                                        FB_Bacnet.StartStopCommand_016.bEnWrite := TRUE;
                                        FB_Bacnet.StartStopCommand_016.bVal := TRUE;
                                    18: 
                                        
                                        FB_Bacnet.StartStopCommand_017.bEnWrite := TRUE;
                                        FB_Bacnet.StartStopCommand_017.bVal := TRUE;
                                    19: 
                                        
                                        FB_Bacnet.StartStopCommand_019.bEnWrite := TRUE;
                                        FB_Bacnet.StartStopCommand_019.bVal := TRUE;
                                    20:
                                        
                                        FB_Bacnet.StartStopCommand_018.bEnWrite := TRUE;
                                        FB_Bacnet.StartStopCommand_018.bVal := TRUE;
                                END_CASE
                            END_IF
                        END_FOR        
                    END_IF
                    // Schedule Unit OFF
                    IF wSchedWEHourEndFG_ = currH AND wSchedWEMinEndFG_ = currM AND NOT bUnitTriggered THEN
                        bUnitTriggered := TRUE;
                        FOR i := 1 TO 20 DO
                            // Send command unit OFF
                            IF bUnitFG_[i] THEN 
                                CASE i OF
                                    1: 
                                        
                                        FB_Bacnet.StartStopCommand_000.bEnWrite := TRUE;
                                        FB_Bacnet.StartStopCommand_000.bVal := FALSE;
                                    2: 
                                        
                                        FB_Bacnet.StartStopCommand_001.bEnWrite := TRUE;
                                        FB_Bacnet.StartStopCommand_001.bVal := FALSE;
                                    3: 
                                        
                                        FB_Bacnet.StartStopCommand_002.bEnWrite := TRUE;
                                        FB_Bacnet.StartStopCommand_002.bVal := FALSE;
                                    4: 
                                        
                                        FB_Bacnet.StartStopCommand_003.bEnWrite := TRUE;
                                        FB_Bacnet.StartStopCommand_003.bVal := FALSE;
                                    5: 
                                        
                                        FB_Bacnet.StartStopCommand_004.bEnWrite := TRUE;
                                        FB_Bacnet.StartStopCommand_004.bVal := FALSE;
                                    6: 
                                        
                                        FB_Bacnet.StartStopCommand_005.bEnWrite := TRUE;
                                        FB_Bacnet.StartStopCommand_005.bVal := FALSE;
                                    7: 
                                        
                                        FB_Bacnet.StartStopCommand_006.bEnWrite := TRUE;
                                        FB_Bacnet.StartStopCommand_006.bVal := FALSE;
                                    8: 
                                        
                                        FB_Bacnet.StartStopCommand_007.bEnWrite := TRUE;
                                        FB_Bacnet.StartStopCommand_007.bVal := FALSE;
                                    9: 
                                        
                                        FB_Bacnet.StartStopCommand_008.bEnWrite := TRUE;
                                        FB_Bacnet.StartStopCommand_008.bVal := FALSE;
                                    10: 
                                        
                                        FB_Bacnet.StartStopCommand_009.bEnWrite := TRUE;
                                        FB_Bacnet.StartStopCommand_009.bVal := FALSE;
                                    11: 
                                        
                                        FB_Bacnet.StartStopCommand_010.bEnWrite := TRUE;
                                        FB_Bacnet.StartStopCommand_010.bVal := FALSE;
                                    12: 
                                        
                                        FB_Bacnet.StartStopCommand_011.bEnWrite := TRUE;
                                        FB_Bacnet.StartStopCommand_011.bVal := FALSE;
                                    13: 
                                        
                                        FB_Bacnet.StartStopCommand_012.bEnWrite := TRUE;
                                        FB_Bacnet.StartStopCommand_012.bVal := FALSE;
                                    14: 
                                        
                                        FB_Bacnet.StartStopCommand_013.bEnWrite := TRUE;
                                        FB_Bacnet.StartStopCommand_013.bVal := FALSE;
                                    15: 
                                        
                                        FB_Bacnet.StartStopCommand_014.bEnWrite := TRUE;
                                        FB_Bacnet.StartStopCommand_014.bVal := FALSE;
                                    16: 
                                        
                                        FB_Bacnet.StartStopCommand_015.bEnWrite := TRUE;
                                        FB_Bacnet.StartStopCommand_015.bVal := FALSE;
                                    17: 
                                        
                                        FB_Bacnet.StartStopCommand_016.bEnWrite := TRUE;
                                        FB_Bacnet.StartStopCommand_016.bVal := FALSE;
                                    18: 
                                        
                                        FB_Bacnet.StartStopCommand_017.bEnWrite := TRUE;
                                        FB_Bacnet.StartStopCommand_017.bVal := FALSE;
                                    19: 
                                        
                                        FB_Bacnet.StartStopCommand_019.bEnWrite := TRUE;
                                        FB_Bacnet.StartStopCommand_019.bVal := FALSE;
                                    20:
                                        
                                        FB_Bacnet.StartStopCommand_018.bEnWrite := TRUE;
                                        FB_Bacnet.StartStopCommand_018.bVal := FALSE;
                                END_CASE
                            END_IF
                        END_FOR
                    END_IF
                END_IF
            END_IF
        END_IF

END_FUNCTION_BLOCK

// ---- POUs/FB_Scheduler/FB_Scheduler_FB2.TcPOU

      FUNCTION_BLOCK FB_Scheduler_FB2
      VAR_INPUT
          currH : WORD;
          currM : WORD;
          currD : WORD;
      END_VAR
      VAR_IN_OUT
          FB_Bacnet : FB_BACnet_DAIKIN_MasterStation_III_No_1;
      END_VAR
      VAR
          i : INT;
          bUnitTriggered : BOOL := FALSE; // New flag to track execution
          prevMinute : WORD := 0;        // New variable to track the previous minute
      END_VAR
      VAR PERSISTENT
          //scheduler var
          bEnSchedFB2_ : BOOL;
          wSchedWDHourStartFB2_ : WORD; 
          wSchedWDMinStartFB2_ : WORD; 
          wSchedWEHourStartFB2_ : WORD; 
          wSchedWEMinStartFB2_ : WORD;
          wSchedWDHourEndFB2_ : WORD;
          wSchedWDMinEndFB2_ : WORD;
          wSchedWEHourEndFB2_ : WORD;
          wSchedWEMinEndFB2_ : WORD;
          //unit var
          bUnitFB2_ : ARRAY [1..13] OF BOOL;
      END_VAR


        // Reset trigger flag at minute change or at the exact scheduled time
        IF currM <> prevMinute OR 
           (currH = wSchedWDHourStartFB2_ AND currM = wSchedWDMinStartFB2_) OR 
           (currH = wSchedWDHourEndFB2_ AND currM = wSchedWDMinEndFB2_) THEN
            bUnitTriggered := FALSE;
            prevMinute := currM;
        END_IF

        // Unit Schedule Enable
        IF bEnSchedFB2_ THEN
            // Weekday schedule
            IF currD >= 1 AND currD <= 5 THEN
                IF (wSchedWDHourStartFB2_ <> wSchedWDHourEndFB2_ OR wSchedWDMinStartFB2_ <> wSchedWDMinEndFB2_) THEN
                    // Schedule Unit ON
                    IF wSchedWDHourStartFB2_ = currH AND wSchedWDMinStartFB2_ = currM AND NOT bUnitTriggered THEN
                        bUnitTriggered := TRUE;
                        FOR i := 1 TO 13 DO
                            // Send command unit ON
                            IF bUnitFB2_[i] THEN 
                                CASE i OF
                                    1: 
                                        
                                        FB_Bacnet.StartStopCommand_037.bEnWrite := TRUE;
                                        FB_Bacnet.StartStopCommand_037.bVal := TRUE;
                                    2: 
                                        
                                        FB_Bacnet.StartStopCommand_038.bEnWrite := TRUE;
                                        FB_Bacnet.StartStopCommand_038.bVal := TRUE;
                                    3: 
                                        
                                        FB_Bacnet.StartStopCommand_039.bEnWrite := TRUE;
                                        FB_Bacnet.StartStopCommand_039.bVal := TRUE;
                                    4: 
                                        //
                                        //FB_Bacnet.StartStopCommand_040.bEnWrite := TRUE;
                                        //FB_Bacnet.StartStopCommand_040.bVal := TRUE;
                                    5: 
                                        
                                        FB_Bacnet.StartStopCommand_041.bEnWrite := TRUE;
                                        FB_Bacnet.StartStopCommand_041.bVal := TRUE;
                                    6: 
                                        
                                        FB_Bacnet.StartStopCommand_042.bEnWrite := TRUE;
                                        FB_Bacnet.StartStopCommand_042.bVal := TRUE;
                                    7: 
                                        
                                        FB_Bacnet.StartStopCommand_043.bEnWrite := TRUE;
                                        FB_Bacnet.StartStopCommand_043.bVal := TRUE;
                                    8: 
                                        //
                                        //FB_Bacnet.StartStopCommand_044.bEnWrite := TRUE;
                                        //FB_Bacnet.StartStopCommand_044.bVal := TRUE;
                                    9: 
                                        
                                        FB_Bacnet.StartStopCommand_045.bEnWrite := TRUE;
                                        FB_Bacnet.StartStopCommand_045.bVal := TRUE;
                                    10: 
                                        
                                        FB_Bacnet.StartStopCommand_046.bEnWrite := TRUE;
                                        FB_Bacnet.StartStopCommand_046.bVal := TRUE;
                                    11: 
                                        //
                                        //FB_Bacnet.StartStopCommand_047.bEnWrite := TRUE;
                                        //FB_Bacnet.StartStopCommand_047.bVal := TRUE;
                                    12: 
                                        //
                                        //FB_Bacnet.StartStopCommand_048.bEnWrite := TRUE;
                                        //FB_Bacnet.StartStopCommand_048.bVal := TRUE;
                                    13: 
                                        
                                        FB_Bacnet.StartStopCommand_049.bEnWrite := TRUE;
                                        FB_Bacnet.StartStopCommand_049.bVal := TRUE;
                                END_CASE
                            END_IF
                        END_FOR
                    END_IF
                    // Schedule Unit OFF
                    IF wSchedWDHourEndFB2_ = currH AND wSchedWDMinEndFB2_ = currM AND NOT bUnitTriggered THEN
                        bUnitTriggered := TRUE;
                        FOR i := 1 TO 13 DO
                            // Send command unit OFF
                            IF bUnitFB2_[i] THEN 
                                CASE i OF
                                    1: 
                                        
                                        FB_Bacnet.StartStopCommand_037.bEnWrite := TRUE;
                                        FB_Bacnet.StartStopCommand_037.bVal := FALSE;
                                    2: 
                                        
                                        FB_Bacnet.StartStopCommand_038.bEnWrite := TRUE;
                                        FB_Bacnet.StartStopCommand_038.bVal := FALSE;
                                    3: 
                                        
                                        FB_Bacnet.StartStopCommand_039.bEnWrite := TRUE;
                                        FB_Bacnet.StartStopCommand_039.bVal := FALSE;
                                    4: 
                                        //
                                        //FB_Bacnet.StartStopCommand_040.bEnWrite := TRUE;
                                        //FB_Bacnet.StartStopCommand_040.bVal := FALSE;
                                    5: 
                                        
                                        FB_Bacnet.StartStopCommand_041.bEnWrite := TRUE;
                                        FB_Bacnet.StartStopCommand_041.bVal := FALSE;
                                    6: 
                                        
                                        FB_Bacnet.StartStopCommand_042.bEnWrite := TRUE;
                                        FB_Bacnet.StartStopCommand_042.bVal := FALSE;
                                    7: 
                                        
                                        FB_Bacnet.StartStopCommand_043.bEnWrite := TRUE;
                                        FB_Bacnet.StartStopCommand_043.bVal := FALSE;
                                    8: 
                                        //
                                        //FB_Bacnet.StartStopCommand_044.bEnWrite := TRUE;
                                        //FB_Bacnet.StartStopCommand_044.bVal := FALSE;
                                    9: 
                                        
                                        FB_Bacnet.StartStopCommand_045.bEnWrite := TRUE;
                                        FB_Bacnet.StartStopCommand_045.bVal := FALSE;
                                    10: 
                                        
                                        FB_Bacnet.StartStopCommand_046.bEnWrite := TRUE;
                                        FB_Bacnet.StartStopCommand_046.bVal := FALSE;
                                    11: 
                                        //
                                        //FB_Bacnet.StartStopCommand_047.bEnWrite := TRUE;
                                        //FB_Bacnet.StartStopCommand_047.bVal := FALSE;
                                    12: 
                                        //
                                        //FB_Bacnet.StartStopCommand_048.bEnWrite := TRUE;
                                        //FB_Bacnet.StartStopCommand_048.bVal := FALSE;
                                    13: 
                                        
                                        FB_Bacnet.StartStopCommand_049.bEnWrite := TRUE;
                                        FB_Bacnet.StartStopCommand_049.bVal := FALSE;
                                END_CASE
                            END_IF
                        END_FOR
                    END_IF
                END_IF
            END_IF

            // Weekend schedule
            IF currD = 0 OR currD = 6 THEN
                IF (wSchedWEHourStartFB2_ <> wSchedWEHourEndFB2_ OR wSchedWEMinStartFB2_ <> wSchedWEMinEndFB2_) THEN
                    // Schedule Unit ON
                    IF wSchedWEHourStartFB2_ = currH AND wSchedWEMinStartFB2_ = currM AND NOT bUnitTriggered THEN
                        bUnitTriggered := TRUE;
                        FOR i := 1 TO 13 DO
                            // Send command unit ON
                            IF bUnitFB2_[i] THEN 
                                CASE i OF
                                    1: 
                                        
                                        FB_Bacnet.StartStopCommand_037.bEnWrite := TRUE;
                                        FB_Bacnet.StartStopCommand_037.bVal := TRUE;
                                    2: 
                                        
                                        FB_Bacnet.StartStopCommand_038.bEnWrite := TRUE;
                                        FB_Bacnet.StartStopCommand_038.bVal := TRUE;
                                    3: 
                                        
                                        FB_Bacnet.StartStopCommand_039.bEnWrite := TRUE;
                                        FB_Bacnet.StartStopCommand_039.bVal := TRUE;
                                    4: 
                                        //
                                        //FB_Bacnet.StartStopCommand_040.bEnWrite := TRUE;
                                        //FB_Bacnet.StartStopCommand_040.bVal := TRUE;
                                    5: 
                                        
                                        FB_Bacnet.StartStopCommand_041.bEnWrite := TRUE;
                                        FB_Bacnet.StartStopCommand_041.bVal := TRUE;
                                    6: 
                                        
                                        FB_Bacnet.StartStopCommand_042.bEnWrite := TRUE;
                                        FB_Bacnet.StartStopCommand_042.bVal := TRUE;
                                    7: 
                                        
                                        FB_Bacnet.StartStopCommand_043.bEnWrite := TRUE;
                                        FB_Bacnet.StartStopCommand_043.bVal := TRUE;
                                    8: 
                                        //
                                        //FB_Bacnet.StartStopCommand_044.bEnWrite := TRUE;
                                        //FB_Bacnet.StartStopCommand_044.bVal := TRUE;
                                    9: 
                                        
                                        FB_Bacnet.StartStopCommand_045.bEnWrite := TRUE;
                                        FB_Bacnet.StartStopCommand_045.bVal := TRUE;
                                    10: 
                                        
                                        FB_Bacnet.StartStopCommand_046.bEnWrite := TRUE;
                                        FB_Bacnet.StartStopCommand_046.bVal := TRUE;
                                    11: 
                                        //
                                        //FB_Bacnet.StartStopCommand_047.bEnWrite := TRUE;
                                        //FB_Bacnet.StartStopCommand_047.bVal := TRUE;
                                    12: 
                                        //
                                        //FB_Bacnet.StartStopCommand_048.bEnWrite := TRUE;
                                        //FB_Bacnet.StartStopCommand_048.bVal := TRUE;
                                    13: 
                                        
                                        FB_Bacnet.StartStopCommand_049.bEnWrite := TRUE;
                                        FB_Bacnet.StartStopCommand_049.bVal := TRUE;
                                END_CASE
                            END_IF
                        END_FOR
                    END_IF
                    // Schedule Unit OFF
                    IF wSchedWEHourEndFB2_ = currH AND wSchedWEMinEndFB2_ = currM AND NOT bUnitTriggered THEN
                        bUnitTriggered := TRUE;
                        FOR i := 1 TO 13 DO
                            // Send command unit OFF
                            IF bUnitFB2_[i] THEN 
                                CASE i OF
                                    1: 
                                        
                                        FB_Bacnet.StartStopCommand_037.bEnWrite := TRUE;
                                        FB_Bacnet.StartStopCommand_037.bVal := FALSE;
                                    2: 
                                        
                                        FB_Bacnet.StartStopCommand_038.bEnWrite := TRUE;
                                        FB_Bacnet.StartStopCommand_038.bVal := FALSE;
                                    3: 
                                        
                                        FB_Bacnet.StartStopCommand_039.bEnWrite := TRUE;
                                        FB_Bacnet.StartStopCommand_039.bVal := FALSE;
                                    4: 
                                        //
                                        //FB_Bacnet.StartStopCommand_040.bEnWrite := TRUE;
                                        //FB_Bacnet.StartStopCommand_040.bVal := FALSE;
                                    5: 
                                        
                                        FB_Bacnet.StartStopCommand_041.bEnWrite := TRUE;
                                        FB_Bacnet.StartStopCommand_041.bVal := FALSE;
                                    6: 
                                        
                                        FB_Bacnet.StartStopCommand_042.bEnWrite := TRUE;
                                        FB_Bacnet.StartStopCommand_042.bVal := FALSE;
                                    7: 
                                        
                                        FB_Bacnet.StartStopCommand_043.bEnWrite := TRUE;
                                        FB_Bacnet.StartStopCommand_043.bVal := FALSE;
                                    8: 
                                        //
                                        //FB_Bacnet.StartStopCommand_044.bEnWrite := TRUE;
                                        //FB_Bacnet.StartStopCommand_044.bVal := FALSE;
                                    9: 
                                        
                                        FB_Bacnet.StartStopCommand_045.bEnWrite := TRUE;
                                        FB_Bacnet.StartStopCommand_045.bVal := FALSE;
                                    10: 
                                        
                                        FB_Bacnet.StartStopCommand_046.bEnWrite := TRUE;
                                        FB_Bacnet.StartStopCommand_046.bVal := FALSE;
                                    11: 
                                        //
                                        //FB_Bacnet.StartStopCommand_047.bEnWrite := TRUE;
                                        //FB_Bacnet.StartStopCommand_047.bVal := FALSE;
                                    12: 
                                        //
                                        //FB_Bacnet.StartStopCommand_048.bEnWrite := TRUE;
                                        //FB_Bacnet.StartStopCommand_048.bVal := FALSE;
                                    13: 
                                        
                                        FB_Bacnet.StartStopCommand_049.bEnWrite := TRUE;
                                        FB_Bacnet.StartStopCommand_049.bVal := FALSE;
                                END_CASE
                            END_IF
                        END_FOR
                    END_IF
                END_IF
            END_IF
        END_IF

END_FUNCTION_BLOCK

// ---- POUs/FB_Scheduler/FB_Scheduler_FB1.TcPOU

      FUNCTION_BLOCK FB_Scheduler_FB1
      VAR_INPUT
          currH : WORD;
          currM : WORD;
          currD : WORD;
      END_VAR
      VAR_IN_OUT
          FB_Bacnet : FB_BACnet_DAIKIN_MasterStation_III_No_1;
      END_VAR
      VAR
          i : INT;
          bUnitTriggered : BOOL := FALSE; // New flag to track execution
          prevMinute : WORD := 0;        // New variable to track the previous minute
      END_VAR
      VAR PERSISTENT
          //scheduler var
          bEnSchedFB1_ : BOOL := FALSE;
          wSchedWDHourStartFB1_ : WORD; 
          wSchedWDMinStartFB1_ : WORD; 
          wSchedWEHourStartFB1_ : WORD; 
          wSchedWEMinStartFB1_ : WORD;
          wSchedWDHourEndFB1_ : WORD;
          wSchedWDMinEndFB1_ : WORD;
          wSchedWEHourEndFB1_ : WORD;
          wSchedWEMinEndFB1_ : WORD;
          //unit var
          bUnitFB1_ : ARRAY [1..17] OF BOOL;
      END_VAR


        // Reset trigger flag at minute change or at the exact scheduled time
        IF currM <> prevMinute OR 
           (currH = wSchedWDHourStartFB1_ AND currM = wSchedWDMinStartFB1_) OR 
           (currH = wSchedWDHourEndFB1_ AND currM = wSchedWDMinEndFB1_) THEN
            bUnitTriggered := FALSE;
            prevMinute := currM;
        END_IF

        // Unit Schedule Enable
        IF bEnSchedFB1_ THEN
            // Weekday schedule
            IF currD >= 1 AND currD <= 5 THEN
                IF (wSchedWDHourStartFB1_ <> wSchedWDHourEndFB1_ OR wSchedWDMinStartFB1_ <> wSchedWDMinEndFB1_) THEN
                    // Schedule Unit ON
                    IF wSchedWDHourStartFB1_ = currH AND wSchedWDMinStartFB1_ = currM AND NOT bUnitTriggered THEN
                        bUnitTriggered := TRUE;
                        FOR i := 1 TO 17 DO
                            // Send command unit ON
                            IF bUnitFB1_[i] THEN 
                                CASE i OF
                                    1: 
                                        
                                        FB_Bacnet.StartStopCommand_020.bEnWrite := TRUE;
                                        FB_Bacnet.StartStopCommand_020.bVal := TRUE;
                                    2: 
                                        
                                        FB_Bacnet.StartStopCommand_021.bEnWrite := TRUE;
                                        FB_Bacnet.StartStopCommand_021.bVal := TRUE;
                                    3: 
                                        
                                        FB_Bacnet.StartStopCommand_022.bEnWrite := TRUE;
                                        FB_Bacnet.StartStopCommand_022.bVal := TRUE;
                                    4: 
                                        
                                        FB_Bacnet.StartStopCommand_023.bEnWrite := TRUE;
                                        FB_Bacnet.StartStopCommand_023.bVal := TRUE;
                                    5: 
                                        
                                        FB_Bacnet.StartStopCommand_024.bEnWrite := TRUE;
                                        FB_Bacnet.StartStopCommand_024.bVal := TRUE;
                                    6: 
                                        
                                        FB_Bacnet.StartStopCommand_025.bEnWrite := TRUE;
                                        FB_Bacnet.StartStopCommand_025.bVal := TRUE;
                                    7: 
                                        
                                        FB_Bacnet.StartStopCommand_026.bEnWrite := TRUE;
                                        FB_Bacnet.StartStopCommand_026.bVal := TRUE;
                                    8: 
                                        
                                        FB_Bacnet.StartStopCommand_027.bEnWrite := TRUE;
                                        FB_Bacnet.StartStopCommand_027.bVal := TRUE;
                                    9: 
                                        
                                        FB_Bacnet.StartStopCommand_028.bEnWrite := TRUE;
                                        FB_Bacnet.StartStopCommand_028.bVal := TRUE;
                                    10: 
                                        
                                        FB_Bacnet.StartStopCommand_029.bEnWrite := TRUE;
                                        FB_Bacnet.StartStopCommand_029.bVal := TRUE;
                                    11: 
                                        
                                        FB_Bacnet.StartStopCommand_030.bEnWrite := TRUE;
                                        FB_Bacnet.StartStopCommand_030.bVal := TRUE;
                                    12: 
                                        
                                        FB_Bacnet.StartStopCommand_031.bEnWrite := TRUE;
                                        FB_Bacnet.StartStopCommand_031.bVal := TRUE;
                                    13: 
                                        
                                        FB_Bacnet.StartStopCommand_032.bEnWrite := TRUE;
                                        FB_Bacnet.StartStopCommand_032.bVal := TRUE;
                                    14: 
                                        
                                        FB_Bacnet.StartStopCommand_033.bEnWrite := TRUE;
                                        FB_Bacnet.StartStopCommand_033.bVal := TRUE;
                                    15: 
                                        
                                        FB_Bacnet.StartStopCommand_034.bEnWrite := TRUE;
                                        FB_Bacnet.StartStopCommand_034.bVal := TRUE;
                                    16: 
                                        
                                        FB_Bacnet.StartStopCommand_035.bEnWrite := TRUE;
                                        FB_Bacnet.StartStopCommand_035.bVal := TRUE;
                                    17: 
                                        
                                        FB_Bacnet.StartStopCommand_036.bEnWrite := TRUE;
                                        FB_Bacnet.StartStopCommand_036.bVal := TRUE;
                                END_CASE
                            END_IF
                        END_FOR
                    END_IF
                    // Schedule Unit OFF
                    IF wSchedWDHourEndFB1_ = currH AND wSchedWDMinEndFB1_ = currM AND NOT bUnitTriggered THEN
                        bUnitTriggered := TRUE;
                        FOR i := 1 TO 17 DO
                            // Send command unit OFF
                            IF bUnitFB1_[i] THEN 
                                CASE i OF
                                    1: 
                                        
                                        FB_Bacnet.StartStopCommand_020.bEnWrite := TRUE;
                                        FB_Bacnet.StartStopCommand_020.bVal := FALSE;
                                    2: 
                                        
                                        FB_Bacnet.StartStopCommand_021.bEnWrite := TRUE;
                                        FB_Bacnet.StartStopCommand_021.bVal := FALSE;
                                    3: 
                                        
                                        FB_Bacnet.StartStopCommand_022.bEnWrite := TRUE;
                                        FB_Bacnet.StartStopCommand_022.bVal := FALSE;
                                    4: 
                                        
                                        FB_Bacnet.StartStopCommand_023.bEnWrite := TRUE;
                                        FB_Bacnet.StartStopCommand_023.bVal := FALSE;
                                    5: 
                                        
                                        FB_Bacnet.StartStopCommand_024.bEnWrite := TRUE;
                                        FB_Bacnet.StartStopCommand_024.bVal := FALSE;
                                    6: 
                                        
                                        FB_Bacnet.StartStopCommand_025.bEnWrite := TRUE;
                                        FB_Bacnet.StartStopCommand_025.bVal := FALSE;
                                    7: 
                                        
                                        FB_Bacnet.StartStopCommand_026.bEnWrite := TRUE;
                                        FB_Bacnet.StartStopCommand_026.bVal := FALSE;
                                    8: 
                                        
                                        FB_Bacnet.StartStopCommand_027.bEnWrite := TRUE;
                                        FB_Bacnet.StartStopCommand_027.bVal := FALSE;
                                    9: 
                                        
                                        FB_Bacnet.StartStopCommand_028.bEnWrite := TRUE;
                                        FB_Bacnet.StartStopCommand_028.bVal := FALSE;
                                    10: 
                                        
                                        FB_Bacnet.StartStopCommand_029.bEnWrite := TRUE;
                                        FB_Bacnet.StartStopCommand_029.bVal := FALSE;
                                    11: 
                                        
                                        FB_Bacnet.StartStopCommand_030.bEnWrite := TRUE;
                                        FB_Bacnet.StartStopCommand_030.bVal := FALSE;
                                    12: 
                                        
                                        FB_Bacnet.StartStopCommand_031.bEnWrite := TRUE;
                                        FB_Bacnet.StartStopCommand_031.bVal := FALSE;
                                    13: 
                                        
                                        FB_Bacnet.StartStopCommand_032.bEnWrite := TRUE;
                                        FB_Bacnet.StartStopCommand_032.bVal := FALSE;
                                    14: 
                                        
                                        FB_Bacnet.StartStopCommand_033.bEnWrite := TRUE;
                                        FB_Bacnet.StartStopCommand_033.bVal := FALSE;
                                    15: 
                                        
                                        FB_Bacnet.StartStopCommand_034.bEnWrite := TRUE;
                                        FB_Bacnet.StartStopCommand_034.bVal := FALSE;
                                    16: 
                                        
                                        FB_Bacnet.StartStopCommand_035.bEnWrite := TRUE;
                                        FB_Bacnet.StartStopCommand_035.bVal := FALSE;
                                    17: 
                                        
                                        FB_Bacnet.StartStopCommand_036.bEnWrite := TRUE;
                                        FB_Bacnet.StartStopCommand_036.bVal := FALSE;
                                END_CASE
                            END_IF
                        END_FOR
                    END_IF
                END_IF
            END_IF

            // Weekend schedule
            IF currD = 0 OR currD = 6 THEN
                IF (wSchedWEHourStartFB1_ <> wSchedWEHourEndFB1_ OR wSchedWEMinStartFB1_ <> wSchedWEMinEndFB1_) THEN
                    // Schedule Unit ON
                    IF wSchedWEHourStartFB1_ = currH AND wSchedWEMinStartFB1_ = currM AND NOT bUnitTriggered THEN
                        bUnitTriggered := TRUE;
                        FOR i := 1 TO 17 DO
                            // Send command unit ON
                            IF bUnitFB1_[i] THEN 
                                CASE i OF
                                    1: 
                                        
                                        FB_Bacnet.StartStopCommand_020.bEnWrite := TRUE;
                                        FB_Bacnet.StartStopCommand_020.bVal := TRUE;
                                    2: 
                                        
                                        FB_Bacnet.StartStopCommand_021.bEnWrite := TRUE;
                                        FB_Bacnet.StartStopCommand_021.bVal := TRUE;
                                    3: 
                                        
                                        FB_Bacnet.StartStopCommand_022.bEnWrite := TRUE;
                                        FB_Bacnet.StartStopCommand_022.bVal := TRUE;
                                    4: 
                                        
                                        FB_Bacnet.StartStopCommand_023.bEnWrite := TRUE;
                                        FB_Bacnet.StartStopCommand_023.bVal := TRUE;
                                    5: 
                                        
                                        FB_Bacnet.StartStopCommand_024.bEnWrite := TRUE;
                                        FB_Bacnet.StartStopCommand_024.bVal := TRUE;
                                    6: 
                                        
                                        FB_Bacnet.StartStopCommand_025.bEnWrite := TRUE;
                                        FB_Bacnet.StartStopCommand_025.bVal := TRUE;
                                    7: 
                                        
                                        FB_Bacnet.StartStopCommand_026.bEnWrite := TRUE;
                                        FB_Bacnet.StartStopCommand_026.bVal := TRUE;
                                    8: 
                                        
                                        FB_Bacnet.StartStopCommand_027.bEnWrite := TRUE;
                                        FB_Bacnet.StartStopCommand_027.bVal := TRUE;
                                    9: 
                                        
                                        FB_Bacnet.StartStopCommand_028.bEnWrite := TRUE;
                                        FB_Bacnet.StartStopCommand_028.bVal := TRUE;
                                    10: 
                                        
                                        FB_Bacnet.StartStopCommand_029.bEnWrite := TRUE;
                                        FB_Bacnet.StartStopCommand_029.bVal := TRUE;
                                    11: 
                                        
                                        FB_Bacnet.StartStopCommand_030.bEnWrite := TRUE;
                                        FB_Bacnet.StartStopCommand_030.bVal := TRUE;
                                    12: 
                                        
                                        FB_Bacnet.StartStopCommand_031.bEnWrite := TRUE;
                                        FB_Bacnet.StartStopCommand_031.bVal := TRUE;
                                    13: 
                                        
                                        FB_Bacnet.StartStopCommand_032.bEnWrite := TRUE;
                                        FB_Bacnet.StartStopCommand_032.bVal := TRUE;
                                    14: 
                                        
                                        FB_Bacnet.StartStopCommand_033.bEnWrite := TRUE;
                                        FB_Bacnet.StartStopCommand_033.bVal := TRUE;
                                    15: 
                                        
                                        FB_Bacnet.StartStopCommand_034.bEnWrite := TRUE;
                                        FB_Bacnet.StartStopCommand_034.bVal := TRUE;
                                    16: 
                                        
                                        FB_Bacnet.StartStopCommand_035.bEnWrite := TRUE;
                                        FB_Bacnet.StartStopCommand_035.bVal := TRUE;
                                    17: 
                                        
                                        FB_Bacnet.StartStopCommand_036.bEnWrite := TRUE;
                                        FB_Bacnet.StartStopCommand_036.bVal := TRUE;
                                END_CASE
                            END_IF
                        END_FOR
                    END_IF
                    // Schedule Unit OFF
                    IF wSchedWEHourEndFB1_ = currH AND wSchedWEMinEndFB1_ = currM AND NOT bUnitTriggered THEN
                        bUnitTriggered := TRUE;
                        FOR i := 1 TO 17 DO
                            // Send command unit OFF
                            IF bUnitFB1_[i] THEN 
                                CASE i OF
                                    1: 
                                        
                                        FB_Bacnet.StartStopCommand_020.bEnWrite := TRUE;
                                        FB_Bacnet.StartStopCommand_020.bVal := FALSE;
                                    2: 
                                        
                                        FB_Bacnet.StartStopCommand_021.bEnWrite := TRUE;
                                        FB_Bacnet.StartStopCommand_021.bVal := FALSE;
                                    3: 
                                        
                                        FB_Bacnet.StartStopCommand_022.bEnWrite := TRUE;
                                        FB_Bacnet.StartStopCommand_022.bVal := FALSE;
                                    4: 
                                        
                                        FB_Bacnet.StartStopCommand_023.bEnWrite := TRUE;
                                        FB_Bacnet.StartStopCommand_023.bVal := FALSE;
                                    5: 
                                        
                                        FB_Bacnet.StartStopCommand_024.bEnWrite := TRUE;
                                        FB_Bacnet.StartStopCommand_024.bVal := FALSE;
                                    6: 
                                        
                                        FB_Bacnet.StartStopCommand_025.bEnWrite := TRUE;
                                        FB_Bacnet.StartStopCommand_025.bVal := FALSE;
                                    7: 
                                        
                                        FB_Bacnet.StartStopCommand_026.bEnWrite := TRUE;
                                        FB_Bacnet.StartStopCommand_026.bVal := FALSE;
                                    8: 
                                        
                                        FB_Bacnet.StartStopCommand_027.bEnWrite := TRUE;
                                        FB_Bacnet.StartStopCommand_027.bVal := FALSE;
                                    9: 
                                        
                                        FB_Bacnet.StartStopCommand_028.bEnWrite := TRUE;
                                        FB_Bacnet.StartStopCommand_028.bVal := FALSE;
                                    10: 
                                        
                                        FB_Bacnet.StartStopCommand_029.bEnWrite := TRUE;
                                        FB_Bacnet.StartStopCommand_029.bVal := FALSE;
                                    11: 
                                        
                                        FB_Bacnet.StartStopCommand_030.bEnWrite := TRUE;
                                        FB_Bacnet.StartStopCommand_030.bVal := FALSE;
                                    12: 
                                        
                                        FB_Bacnet.StartStopCommand_031.bEnWrite := TRUE;
                                        FB_Bacnet.StartStopCommand_031.bVal := FALSE;
                                    13: 
                                        
                                        FB_Bacnet.StartStopCommand_032.bEnWrite := TRUE;
                                        FB_Bacnet.StartStopCommand_032.bVal := FALSE;
                                    14: 
                                        
                                        FB_Bacnet.StartStopCommand_033.bEnWrite := TRUE;
                                        FB_Bacnet.StartStopCommand_033.bVal := FALSE;
                                    15: 
                                        
                                        FB_Bacnet.StartStopCommand_034.bEnWrite := TRUE;
                                        FB_Bacnet.StartStopCommand_034.bVal := FALSE;
                                    16: 
                                        
                                        FB_Bacnet.StartStopCommand_035.bEnWrite := TRUE;
                                        FB_Bacnet.StartStopCommand_035.bVal := FALSE;
                                    17: 
                                        
                                        FB_Bacnet.StartStopCommand_036.bEnWrite := TRUE;
                                        FB_Bacnet.StartStopCommand_036.bVal := FALSE;
                                END_CASE
                            END_IF
                        END_FOR
                    END_IF
                END_IF
            END_IF
        END_IF

END_FUNCTION_BLOCK

// ---- POUs/FB_Scheduler/FB_Scheduler_FMZ.TcPOU

      FUNCTION_BLOCK FB_Scheduler_FMZ
      VAR_INPUT
          currH : WORD;
          currM : WORD;
          currD : WORD;
      END_VAR
      VAR_IN_OUT
          FB_Bacnet : FB_BACnet_DAIKIN_MasterStation_III_No_1;
      END_VAR
      VAR
          i : INT;
          bUnitTriggered : BOOL := FALSE; // Flag to track execution
          prevMinute : WORD := 0;        // Track previous minute
      END_VAR
      VAR PERSISTENT
          //scheduler var
          bEnSchedFMZ_ : BOOL := FALSE;
          wSchedWDHourStartFMZ_ : WORD; 
          wSchedWDMinStartFMZ_ : WORD; 
          wSchedWEHourStartFMZ_ : WORD; 
          wSchedWEMinStartFMZ_ : WORD;
          wSchedWDHourEndFMZ_ : WORD;
          wSchedWDMinEndFMZ_ : WORD; 
          wSchedWEHourEndFMZ_ : WORD; 
          wSchedWEMinEndFMZ_ : WORD;
          //unit var
          bUnitFMZ_ : ARRAY [1..21] OF BOOL;
      END_VAR


        // Reset trigger flag at minute change or at the exact scheduled time
        IF currM <> prevMinute OR 
           (currH = wSchedWDHourStartFMZ_ AND currM = wSchedWDMinStartFMZ_) OR 
           (currH = wSchedWDHourEndFMZ_ AND currM = wSchedWDMinEndFMZ_) THEN
            bUnitTriggered := FALSE;
            prevMinute := currM;
        END_IF

        // Unit Schedule Enable
        IF bEnSchedFMZ_ THEN
            // Weekday schedule
            IF currD >= 1 AND currD <= 5 THEN
                IF (wSchedWDHourStartFMZ_ <> wSchedWDHourEndFMZ_ OR wSchedWDMinStartFMZ_ <> wSchedWDMinEndFMZ_) THEN
                    // Schedule Unit ON
                    IF wSchedWDHourStartFMZ_ = currH AND wSchedWDMinStartFMZ_ = currM AND NOT bUnitTriggered THEN
                        bUnitTriggered := TRUE;
                        FOR i := 1 TO 21 DO
                            // Send command unit ON
                            IF bUnitFMZ_[i] THEN 
                                CASE i OF
                                    1: 
                                        
                                        FB_Bacnet.StartStopCommand_064.bEnWrite := TRUE;
                                        FB_Bacnet.StartStopCommand_064.bVal := TRUE;
                                    2: 
                                        
                                        FB_Bacnet.StartStopCommand_065.bEnWrite := TRUE;
                                        FB_Bacnet.StartStopCommand_065.bVal := TRUE;
                                    3: 
                                        
                                        FB_Bacnet.StartStopCommand_066.bEnWrite := TRUE;
                                        FB_Bacnet.StartStopCommand_066.bVal := TRUE;
                                    4: 
                                        
                                        FB_Bacnet.StartStopCommand_067.bEnWrite := TRUE;
                                        FB_Bacnet.StartStopCommand_067.bVal := TRUE;
                                    5: 
                                        
                                        FB_Bacnet.StartStopCommand_068.bEnWrite := TRUE;
                                        FB_Bacnet.StartStopCommand_068.bVal := TRUE;
                                    6: 
                                        
                                        FB_Bacnet.StartStopCommand_069.bEnWrite := TRUE;
                                        FB_Bacnet.StartStopCommand_069.bVal := TRUE;
                                    7: 
                                        
                                        FB_Bacnet.StartStopCommand_070.bEnWrite := TRUE;
                                        FB_Bacnet.StartStopCommand_070.bVal := TRUE;
                                    8: 
                                        
                                        FB_Bacnet.StartStopCommand_071.bEnWrite := TRUE;
                                        FB_Bacnet.StartStopCommand_071.bVal := TRUE;
                                    9: 
                                        
                                        FB_Bacnet.StartStopCommand_072.bEnWrite := TRUE;
                                        FB_Bacnet.StartStopCommand_072.bVal := TRUE;
                                    10: 
                                        
                                        FB_Bacnet.StartStopCommand_073.bEnWrite := TRUE;
                                        FB_Bacnet.StartStopCommand_073.bVal := TRUE;
                                    11: 
                                        
                                        FB_Bacnet.StartStopCommand_074.bEnWrite := TRUE;
                                        FB_Bacnet.StartStopCommand_074.bVal := TRUE;
                                    12: 
                                        
                                        FB_Bacnet.StartStopCommand_075.bEnWrite := TRUE;
                                        FB_Bacnet.StartStopCommand_075.bVal := TRUE;
                                    13: 
                                        
                                        FB_Bacnet.StartStopCommand_076.bEnWrite := TRUE;
                                        FB_Bacnet.StartStopCommand_076.bVal := TRUE;
                                    14: 
                                        
                                        FB_Bacnet.StartStopCommand_077.bEnWrite := TRUE;
                                        FB_Bacnet.StartStopCommand_077.bVal := TRUE;
                                    15: 
                                        
                                        FB_Bacnet.StartStopCommand_078.bEnWrite := TRUE;
                                        FB_Bacnet.StartStopCommand_078.bVal := TRUE;
                                    16: 
                                        
                                        FB_Bacnet.StartStopCommand_079.bEnWrite := TRUE;
                                        FB_Bacnet.StartStopCommand_079.bVal := TRUE;
                                    17: 
                                        
                                        FB_Bacnet.StartStopCommand_080.bEnWrite := TRUE;
                                        FB_Bacnet.StartStopCommand_080.bVal := TRUE;
                                    18: 
                                        
                                        FB_Bacnet.StartStopCommand_081.bEnWrite := TRUE;
                                        FB_Bacnet.StartStopCommand_081.bVal := TRUE;
                                    19: 
                                        
                                        FB_Bacnet.StartStopCommand_082.bEnWrite := TRUE;
                                        FB_Bacnet.StartStopCommand_082.bVal := TRUE;
                                    20: 
                                        
                                        FB_Bacnet.StartStopCommand_083.bEnWrite := TRUE;
                                        FB_Bacnet.StartStopCommand_083.bVal := TRUE;
                                    21: 
                                        
                                        FB_Bacnet.StartStopCommand_084.bEnWrite := TRUE;
                                        FB_Bacnet.StartStopCommand_084.bVal := TRUE;
                                END_CASE
                            END_IF
                        END_FOR
                    END_IF
                    // Schedule Unit OFF
                    IF wSchedWDHourEndFMZ_ = currH AND wSchedWDMinEndFMZ_ = currM AND NOT bUnitTriggered THEN
                        bUnitTriggered := TRUE;
                        FOR i := 1 TO 21 DO
                            // Send command unit OFF
                            IF bUnitFMZ_[i] THEN 
                                CASE i OF
                                    1: 
                                        
                                        FB_Bacnet.StartStopCommand_064.bEnWrite := TRUE;
                                        FB_Bacnet.StartStopCommand_064.bVal := FALSE;
                                    2: 
                                        
                                        FB_Bacnet.StartStopCommand_065.bEnWrite := TRUE;
                                        FB_Bacnet.StartStopCommand_065.bVal := FALSE;
                                    3: 
                                        
                                        FB_Bacnet.StartStopCommand_066.bEnWrite := TRUE;
                                        FB_Bacnet.StartStopCommand_066.bVal := FALSE;
                                    4: 
                                        
                                        FB_Bacnet.StartStopCommand_067.bEnWrite := TRUE;
                                        FB_Bacnet.StartStopCommand_067.bVal := FALSE;
                                    5: 
                                        
                                        FB_Bacnet.StartStopCommand_068.bEnWrite := TRUE;
                                        FB_Bacnet.StartStopCommand_068.bVal := FALSE;
                                    6: 
                                        
                                        FB_Bacnet.StartStopCommand_069.bEnWrite := TRUE;
                                        FB_Bacnet.StartStopCommand_069.bVal := FALSE;
                                    7: 
                                        
                                        FB_Bacnet.StartStopCommand_070.bEnWrite := TRUE;
                                        FB_Bacnet.StartStopCommand_070.bVal := FALSE;
                                    8: 
                                        
                                        FB_Bacnet.StartStopCommand_071.bEnWrite := TRUE;
                                        FB_Bacnet.StartStopCommand_071.bVal := FALSE;
                                    9: 
                                        
                                        FB_Bacnet.StartStopCommand_072.bEnWrite := TRUE;
                                        FB_Bacnet.StartStopCommand_072.bVal := FALSE;
                                    10: 
                                        
                                        FB_Bacnet.StartStopCommand_073.bEnWrite := TRUE;
                                        FB_Bacnet.StartStopCommand_073.bVal := FALSE;
                                    11: 
                                        
                                        FB_Bacnet.StartStopCommand_074.bEnWrite := TRUE;
                                        FB_Bacnet.StartStopCommand_074.bVal := FALSE;
                                    12: 
                                        
                                        FB_Bacnet.StartStopCommand_075.bEnWrite := TRUE;
                                        FB_Bacnet.StartStopCommand_075.bVal := FALSE;
                                    13: 
                                        
                                        FB_Bacnet.StartStopCommand_076.bEnWrite := TRUE;
                                        FB_Bacnet.StartStopCommand_076.bVal := FALSE;
                                    14: 
                                        
                                        FB_Bacnet.StartStopCommand_077.bEnWrite := TRUE;
                                        FB_Bacnet.StartStopCommand_077.bVal := FALSE;
                                    15: 
                                        
                                        FB_Bacnet.StartStopCommand_078.bEnWrite := TRUE;
                                        FB_Bacnet.StartStopCommand_078.bVal := FALSE;
                                    16: 
                                        
                                        FB_Bacnet.StartStopCommand_079.bEnWrite := TRUE;
                                        FB_Bacnet.StartStopCommand_079.bVal := FALSE;
                                    17: 
                                        
                                        FB_Bacnet.StartStopCommand_080.bEnWrite := TRUE;
                                        FB_Bacnet.StartStopCommand_080.bVal := FALSE;
                                    18: 
                                        
                                        FB_Bacnet.StartStopCommand_081.bEnWrite := TRUE;
                                        FB_Bacnet.StartStopCommand_081.bVal := FALSE;
                                    19: 
                                        
                                        FB_Bacnet.StartStopCommand_082.bEnWrite := TRUE;
                                        FB_Bacnet.StartStopCommand_082.bVal := FALSE;
                                    20: 
                                        
                                        FB_Bacnet.StartStopCommand_083.bEnWrite := TRUE;
                                        FB_Bacnet.StartStopCommand_083.bVal := FALSE;
                                    21: 
                                        
                                        FB_Bacnet.StartStopCommand_084.bEnWrite := TRUE;
                                        FB_Bacnet.StartStopCommand_084.bVal := FALSE;
                                END_CASE
                            END_IF
                        END_FOR
                    END_IF
                END_IF
            END_IF

            // Weekend schedule
            IF currD = 0 OR currD = 6 THEN
                IF (wSchedWEHourStartFMZ_ <> wSchedWEHourEndFMZ_ OR wSchedWEMinStartFMZ_ <> wSchedWEMinEndFMZ_) THEN
                    // Schedule Unit ON
                    IF wSchedWEHourStartFMZ_ = currH AND wSchedWEMinStartFMZ_ = currM AND NOT bUnitTriggered THEN
                        bUnitTriggered := TRUE;
                        FOR i := 1 TO 21 DO
                            // Send command unit ON
                            IF bUnitFMZ_[i] THEN 
                                CASE i OF
                                    1: 
                                        
                                        FB_Bacnet.StartStopCommand_064.bEnWrite := TRUE;
                                        FB_Bacnet.StartStopCommand_064.bVal := TRUE;
                                    2: 
                                        
                                        FB_Bacnet.StartStopCommand_065.bEnWrite := TRUE;
                                        FB_Bacnet.StartStopCommand_065.bVal := TRUE;
                                    3: 
                                        
                                        FB_Bacnet.StartStopCommand_066.bEnWrite := TRUE;
                                        FB_Bacnet.StartStopCommand_066.bVal := TRUE;
                                    4: 
                                        
                                        FB_Bacnet.StartStopCommand_067.bEnWrite := TRUE;
                                        FB_Bacnet.StartStopCommand_067.bVal := TRUE;
                                    5: 
                                        
                                        FB_Bacnet.StartStopCommand_068.bEnWrite := TRUE;
                                        FB_Bacnet.StartStopCommand_068.bVal := TRUE;
                                    6: 
                                        
                                        FB_Bacnet.StartStopCommand_069.bEnWrite := TRUE;
                                        FB_Bacnet.StartStopCommand_069.bVal := TRUE;
                                    7: 
                                        
                                        FB_Bacnet.StartStopCommand_070.bEnWrite := TRUE;
                                        FB_Bacnet.StartStopCommand_070.bVal := TRUE;
                                    8: 
                                        
                                        FB_Bacnet.StartStopCommand_071.bEnWrite := TRUE;
                                        FB_Bacnet.StartStopCommand_071.bVal := TRUE;
                                    9: 
                                        
                                        FB_Bacnet.StartStopCommand_072.bEnWrite := TRUE;
                                        FB_Bacnet.StartStopCommand_072.bVal := TRUE;
                                    10: 
                                        
                                        FB_Bacnet.StartStopCommand_073.bEnWrite := TRUE;
                                        FB_Bacnet.StartStopCommand_073.bVal := TRUE;
                                    11: 
                                        
                                        FB_Bacnet.StartStopCommand_074.bEnWrite := TRUE;
                                        FB_Bacnet.StartStopCommand_074.bVal := TRUE;
                                    12: 
                                        
                                        FB_Bacnet.StartStopCommand_075.bEnWrite := TRUE;
                                        FB_Bacnet.StartStopCommand_075.bVal := TRUE;
                                    13: 
                                        
                                        FB_Bacnet.StartStopCommand_076.bEnWrite := TRUE;
                                        FB_Bacnet.StartStopCommand_076.bVal := TRUE;
                                    14: 
                                        
                                        FB_Bacnet.StartStopCommand_077.bEnWrite := TRUE;
                                        FB_Bacnet.StartStopCommand_077.bVal := TRUE;
                                    15: 
                                        
                                        FB_Bacnet.StartStopCommand_078.bEnWrite := TRUE;
                                        FB_Bacnet.StartStopCommand_078.bVal := TRUE;
                                    16: 
                                        
                                        FB_Bacnet.StartStopCommand_079.bEnWrite := TRUE;
                                        FB_Bacnet.StartStopCommand_079.bVal := TRUE;
                                    17: 
                                        
                                        FB_Bacnet.StartStopCommand_080.bEnWrite := TRUE;
                                        FB_Bacnet.StartStopCommand_080.bVal := TRUE;
                                    18: 
                                        
                                        FB_Bacnet.StartStopCommand_081.bEnWrite := TRUE;
                                        FB_Bacnet.StartStopCommand_081.bVal := TRUE;
                                    19: 
                                        
                                        FB_Bacnet.StartStopCommand_082.bEnWrite := TRUE;
                                        FB_Bacnet.StartStopCommand_082.bVal := TRUE;
                                    20: 
                                        
                                        FB_Bacnet.StartStopCommand_083.bEnWrite := TRUE;
                                        FB_Bacnet.StartStopCommand_083.bVal := TRUE;
                                    21: 
                                        
                                        FB_Bacnet.StartStopCommand_084.bEnWrite := TRUE;
                                        FB_Bacnet.StartStopCommand_084.bVal := TRUE;
                                END_CASE
                            END_IF
                        END_FOR
                    END_IF
                    // Schedule Unit OFF
                    IF wSchedWEHourEndFMZ_ = currH AND wSchedWEMinEndFMZ_ = currM AND NOT bUnitTriggered THEN
                        bUnitTriggered := TRUE;
                        FOR i := 1 TO 21 DO
                            // Send command unit OFF
                            IF bUnitFMZ_[i] THEN 
                                CASE i OF
                                    1: 
                                        
                                        FB_Bacnet.StartStopCommand_064.bEnWrite := TRUE;
                                        FB_Bacnet.StartStopCommand_064.bVal := FALSE;
                                    2: 
                                        
                                        FB_Bacnet.StartStopCommand_065.bEnWrite := TRUE;
                                        FB_Bacnet.StartStopCommand_065.bVal := FALSE;
                                    3: 
                                        
                                        FB_Bacnet.StartStopCommand_066.bEnWrite := TRUE;
                                        FB_Bacnet.StartStopCommand_066.bVal := FALSE;
                                    4: 
                                        
                                        FB_Bacnet.StartStopCommand_067.bEnWrite := TRUE;
                                        FB_Bacnet.StartStopCommand_067.bVal := FALSE;
                                    5: 
                                        
                                        FB_Bacnet.StartStopCommand_068.bEnWrite := TRUE;
                                        FB_Bacnet.StartStopCommand_068.bVal := FALSE;
                                    6: 
                                        
                                        FB_Bacnet.StartStopCommand_069.bEnWrite := TRUE;
                                        FB_Bacnet.StartStopCommand_069.bVal := FALSE;
                                    7: 
                                        
                                        FB_Bacnet.StartStopCommand_070.bEnWrite := TRUE;
                                        FB_Bacnet.StartStopCommand_070.bVal := FALSE;
                                    8: 
                                        
                                        FB_Bacnet.StartStopCommand_071.bEnWrite := TRUE;
                                        FB_Bacnet.StartStopCommand_071.bVal := FALSE;
                                    9: 
                                        
                                        FB_Bacnet.StartStopCommand_072.bEnWrite := TRUE;
                                        FB_Bacnet.StartStopCommand_072.bVal := FALSE;
                                    10: 
                                        
                                        FB_Bacnet.StartStopCommand_073.bEnWrite := TRUE;
                                        FB_Bacnet.StartStopCommand_073.bVal := FALSE;
                                    11: 
                                        
                                        FB_Bacnet.StartStopCommand_074.bEnWrite := TRUE;
                                        FB_Bacnet.StartStopCommand_074.bVal := FALSE;
                                    12: 
                                        
                                        FB_Bacnet.StartStopCommand_075.bEnWrite := TRUE;
                                        FB_Bacnet.StartStopCommand_075.bVal := FALSE;
                                    13: 
                                        
                                        FB_Bacnet.StartStopCommand_076.bEnWrite := TRUE;
                                        FB_Bacnet.StartStopCommand_076.bVal := FALSE;
                                    14: 
                                        
                                        FB_Bacnet.StartStopCommand_077.bEnWrite := TRUE;
                                        FB_Bacnet.StartStopCommand_077.bVal := FALSE;
                                    15: 
                                        
                                        FB_Bacnet.StartStopCommand_078.bEnWrite := TRUE;
                                        FB_Bacnet.StartStopCommand_078.bVal := FALSE;
                                    16: 
                                        
                                        FB_Bacnet.StartStopCommand_079.bEnWrite := TRUE;
                                        FB_Bacnet.StartStopCommand_079.bVal := FALSE;
                                    17: 
                                        
                                        FB_Bacnet.StartStopCommand_080.bEnWrite := TRUE;
                                        FB_Bacnet.StartStopCommand_080.bVal := FALSE;
                                    18: 
                                        
                                        FB_Bacnet.StartStopCommand_081.bEnWrite := TRUE;
                                        FB_Bacnet.StartStopCommand_081.bVal := FALSE;
                                    19: 
                                        
                                        FB_Bacnet.StartStopCommand_082.bEnWrite := TRUE;
                                        FB_Bacnet.StartStopCommand_082.bVal := FALSE;
                                    20: 
                                        
                                        FB_Bacnet.StartStopCommand_083.bEnWrite := TRUE;
                                        FB_Bacnet.StartStopCommand_083.bVal := FALSE;
                                    21: 
                                        
                                        FB_Bacnet.StartStopCommand_084.bEnWrite := TRUE;
                                        FB_Bacnet.StartStopCommand_084.bVal := FALSE;
                                END_CASE
                            END_IF
                        END_FOR
                    END_IF
                END_IF
            END_IF
        END_IF

END_FUNCTION_BLOCK

// ---- POUs/FB_Scheduler/FB_Scheduler_FMZ2.TcPOU

      FUNCTION_BLOCK FB_Scheduler_FMZ2
      VAR_INPUT
          currH : WORD;
          currM : WORD;
          currD : WORD;
      END_VAR
      VAR_IN_OUT
          FB_Bacnet : FB_BACnet_DAIKIN_MasterStation_III_No_1;
      END_VAR
      VAR
          i : INT;
          bUnitTriggered : BOOL := FALSE; // New flag to track execution
          prevMinute : WORD := 0;        // New variable to track the previous minute
      END_VAR
      VAR PERSISTENT
          //scheduler var
          bEnSchedFMZ2_ : BOOL := FALSE;
          wSchedWDHourStartFMZ2_ : WORD; 
          wSchedWDMinStartFMZ2_ : WORD; 
          wSchedWEHourStartFMZ2_ : WORD; 
          wSchedWEMinStartFMZ2_ : WORD;
          wSchedWDHourEndFMZ2_ : WORD;
          wSchedWDMinEndFMZ2_ : WORD;
          wSchedWEHourEndFMZ2_ : WORD;
          wSchedWEMinEndFMZ2_ : WORD;
          //unit var
          bUnitFMZ2_ : ARRAY [1..8] OF BOOL;
      END_VAR


        // Reset trigger flag at minute change or at the exact scheduled time
        IF currM <> prevMinute OR 
           (currH = wSchedWDHourStartFMZ2_ AND currM = wSchedWDMinStartFMZ2_) OR 
           (currH = wSchedWDHourEndFMZ2_ AND currM = wSchedWDMinEndFMZ2_) THEN
            bUnitTriggered := FALSE;
            prevMinute := currM;
        END_IF

        // Unit Schedule Enable
        IF bEnSchedFMZ2_ THEN
            // Weekday schedule
            IF currD >= 1 AND currD <= 5 THEN
                IF (wSchedWDHourStartFMZ2_ <> wSchedWDHourEndFMZ2_ OR wSchedWDMinStartFMZ2_ <> wSchedWDMinEndFMZ2_) THEN
                    // Schedule Unit ON
                    IF wSchedWDHourStartFMZ2_ = currH AND wSchedWDMinStartFMZ2_ = currM AND NOT bUnitTriggered THEN
                        bUnitTriggered := TRUE;
                        FOR i := 1 TO 8 DO
                            // Send command unit ON
                            IF bUnitFMZ2_[i] THEN 
                                CASE i OF
                                    1: FB_Bacnet.StartStopCommand_096.bEnWrite := TRUE;
                                       FB_Bacnet.StartStopCommand_096.bVal := TRUE;
                                    2: FB_Bacnet.StartStopCommand_097.bEnWrite := TRUE;
                                       FB_Bacnet.StartStopCommand_097.bVal := TRUE;
                                    3: FB_Bacnet.StartStopCommand_098.bEnWrite := TRUE;
                                       FB_Bacnet.StartStopCommand_098.bVal := TRUE;
                                    4: FB_Bacnet.StartStopCommand_099.bEnWrite := TRUE;
                                       FB_Bacnet.StartStopCommand_099.bVal := TRUE;
                                    5: FB_Bacnet.StartStopCommand_100.bEnWrite := TRUE;
                                       FB_Bacnet.StartStopCommand_100.bVal := TRUE;
                                    6: FB_Bacnet.StartStopCommand_101.bEnWrite := TRUE;
                                       FB_Bacnet.StartStopCommand_101.bVal := TRUE;
                                    7: FB_Bacnet.StartStopCommand_102.bEnWrite := TRUE;
                                       FB_Bacnet.StartStopCommand_102.bVal := TRUE;
                                    8: FB_Bacnet.StartStopCommand_103.bEnWrite := TRUE;
                                       FB_Bacnet.StartStopCommand_103.bVal := TRUE;
                                END_CASE
                            END_IF
                        END_FOR
                    END_IF
                    // Schedule Unit OFF
                    IF wSchedWDHourEndFMZ2_ = currH AND wSchedWDMinEndFMZ2_ = currM AND NOT bUnitTriggered THEN
                        bUnitTriggered := TRUE;
                        FOR i := 1 TO 8 DO
                            // Send command unit OFF
                            IF bUnitFMZ2_[i] THEN 
                                CASE i OF
                                    1: FB_Bacnet.StartStopCommand_096.bEnWrite := TRUE;
                                       FB_Bacnet.StartStopCommand_096.bVal := FALSE;
                                    2: FB_Bacnet.StartStopCommand_097.bEnWrite := TRUE;
                                       FB_Bacnet.StartStopCommand_097.bVal := FALSE;
                                    3: FB_Bacnet.StartStopCommand_098.bEnWrite := TRUE;
                                       FB_Bacnet.StartStopCommand_098.bVal := FALSE;
                                    4: FB_Bacnet.StartStopCommand_099.bEnWrite := TRUE;
                                       FB_Bacnet.StartStopCommand_099.bVal := FALSE;
                                    5: FB_Bacnet.StartStopCommand_100.bEnWrite := TRUE;
                                       FB_Bacnet.StartStopCommand_100.bVal := FALSE;
                                    6: FB_Bacnet.StartStopCommand_101.bEnWrite := TRUE;
                                       FB_Bacnet.StartStopCommand_101.bVal := FALSE;
                                    7: FB_Bacnet.StartStopCommand_102.bEnWrite := TRUE;
                                       FB_Bacnet.StartStopCommand_102.bVal := FALSE;
                                    8: FB_Bacnet.StartStopCommand_103.bEnWrite := TRUE;
                                       FB_Bacnet.StartStopCommand_103.bVal := FALSE;
                                END_CASE
                            END_IF
                        END_FOR
                    END_IF
                END_IF
            END_IF

            // Weekend schedule
            IF currD = 0 OR currD = 6 THEN
                IF (wSchedWEHourStartFMZ2_ <> wSchedWEHourEndFMZ2_ OR wSchedWEMinStartFMZ2_ <> wSchedWEMinEndFMZ2_) THEN
                    // Schedule Unit ON
                    IF wSchedWEHourStartFMZ2_ = currH AND wSchedWEMinStartFMZ2_ = currM AND NOT bUnitTriggered THEN
                        bUnitTriggered := TRUE;
                        FOR i := 1 TO 8 DO
                            // Send command unit ON
                            IF bUnitFMZ2_[i] THEN 
                                CASE i OF
                                    1: FB_Bacnet.StartStopCommand_096.bEnWrite := TRUE;
                                       FB_Bacnet.StartStopCommand_096.bVal := TRUE;
                                    2: FB_Bacnet.StartStopCommand_097.bEnWrite := TRUE;
                                       FB_Bacnet.StartStopCommand_097.bVal := TRUE;
                                    3: FB_Bacnet.StartStopCommand_098.bEnWrite := TRUE;
                                       FB_Bacnet.StartStopCommand_098.bVal := TRUE;
                                    4: FB_Bacnet.StartStopCommand_099.bEnWrite := TRUE;
                                       FB_Bacnet.StartStopCommand_099.bVal := TRUE;
                                    5: FB_Bacnet.StartStopCommand_100.bEnWrite := TRUE;
                                       FB_Bacnet.StartStopCommand_100.bVal := TRUE;
                                    6: FB_Bacnet.StartStopCommand_101.bEnWrite := TRUE;
                                       FB_Bacnet.StartStopCommand_101.bVal := TRUE;
                                    7: FB_Bacnet.StartStopCommand_102.bEnWrite := TRUE;
                                       FB_Bacnet.StartStopCommand_102.bVal := TRUE;
                                    8: FB_Bacnet.StartStopCommand_103.bEnWrite := TRUE;
                                       FB_Bacnet.StartStopCommand_103.bVal := TRUE;
                                END_CASE
                            END_IF
                        END_FOR
                    END_IF
                    // Schedule Unit OFF
                    IF wSchedWEHourEndFMZ2_ = currH AND wSchedWEMinEndFMZ2_ = currM AND NOT bUnitTriggered THEN
                        bUnitTriggered := TRUE;
                        FOR i := 1 TO 8 DO
                            // Send command unit OFF
                            IF bUnitFMZ2_[i] THEN 
                                CASE i OF
                                    1: FB_Bacnet.StartStopCommand_096.bEnWrite := TRUE;
                                       FB_Bacnet.StartStopCommand_096.bVal := FALSE;
                                    2: FB_Bacnet.StartStopCommand_097.bEnWrite := TRUE;
                                       FB_Bacnet.StartStopCommand_097.bVal := FALSE;
                                    3: FB_Bacnet.StartStopCommand_098.bEnWrite := TRUE;
                                       FB_Bacnet.StartStopCommand_098.bVal := FALSE;
                                    4: FB_Bacnet.StartStopCommand_099.bEnWrite := TRUE;
                                       FB_Bacnet.StartStopCommand_099.bVal := FALSE;
                                    5: FB_Bacnet.StartStopCommand_100.bEnWrite := TRUE;
                                       FB_Bacnet.StartStopCommand_100.bVal := FALSE;
                                    6: FB_Bacnet.StartStopCommand_101.bEnWrite := TRUE;
                                       FB_Bacnet.StartStopCommand_101.bVal := FALSE;
                                    7: FB_Bacnet.StartStopCommand_102.bEnWrite := TRUE;
                                       FB_Bacnet.StartStopCommand_102.bVal := FALSE;
                                    8: FB_Bacnet.StartStopCommand_103.bEnWrite := TRUE;
                                       FB_Bacnet.StartStopCommand_103.bVal := FALSE;
                                END_CASE
                            END_IF
                        END_FOR
                    END_IF
                END_IF
            END_IF
        END_IF

END_FUNCTION_BLOCK

// ---- POUs/FB_Scheduler/FB_Scheduler_F2.TcPOU

      FUNCTION_BLOCK FB_Scheduler_F2
      VAR_INPUT
          currH : WORD;
          currM : WORD;
          currD : WORD;
      END_VAR
      VAR_IN_OUT
          FB_Bacnet : FB_BACnet_DAIKIN_MasterStation_III_No_1;
      END_VAR
      VAR
          i : INT;
          bUnitTriggered : BOOL := FALSE; // New flag to track execution
          prevMinute : WORD := 0;        // New variable to track the previous minute
      END_VAR
      VAR PERSISTENT
          //scheduler var
          bEnSchedF2_ : BOOL := FALSE;
          wSchedWDHourStartF2_ : WORD; 
          wSchedWDMinStartF2_ : WORD; 
          wSchedWEHourStartF2_ : WORD; 
          wSchedWEMinStartF2_ : WORD;
          wSchedWDHourEndF2_ : WORD;
          wSchedWDMinEndF2_ : WORD;
          wSchedWEHourEndF2_ : WORD;
          wSchedWEMinEndF2_ : WORD;
          //unit var
          bUnitF2_ : ARRAY [1..23] OF BOOL;
      END_VAR


        // Reset trigger flag at minute change or at the exact scheduled time
        IF currM <> prevMinute OR 
           (currH = wSchedWDHourStartF2_ AND currM = wSchedWDMinStartF2_) OR 
           (currH = wSchedWDHourEndF2_ AND currM = wSchedWDMinEndF2_) THEN
            bUnitTriggered := FALSE;
            prevMinute := currM;
        END_IF

        // Unit Schedule Enable
        IF bEnSchedF2_ THEN
            // Weekday schedule
            IF currD >= 1 AND currD <= 5 THEN
                IF (wSchedWDHourStartF2_ <> wSchedWDHourEndF2_ OR wSchedWDMinStartF2_ <> wSchedWDMinEndF2_) THEN
                    // Schedule Unit ON
                    IF wSchedWDHourStartF2_ = currH AND wSchedWDMinStartF2_ = currM AND NOT bUnitTriggered THEN
                        bUnitTriggered := TRUE;
                        FOR i := 1 TO 23 DO
                            // Send command unit ON
                            IF bUnitF2_[i] THEN 
                                CASE i OF
                                    1: 
                                        
                                        FB_Bacnet.StartStopCommand_128.bEnWrite := TRUE;
                                        FB_Bacnet.StartStopCommand_128.bVal := TRUE;
                                    2: 
                                        
                                        FB_Bacnet.StartStopCommand_129.bEnWrite := TRUE;
                                        FB_Bacnet.StartStopCommand_129.bVal := TRUE;
                                    3: 
                                        
                                        FB_Bacnet.StartStopCommand_130.bEnWrite := TRUE;
                                        FB_Bacnet.StartStopCommand_130.bVal := TRUE;
                                    4: 
                                        
                                        FB_Bacnet.StartStopCommand_131.bEnWrite := TRUE;
                                        FB_Bacnet.StartStopCommand_131.bVal := TRUE;
                                    5: 
                                        
                                        FB_Bacnet.StartStopCommand_132.bEnWrite := TRUE;
                                        FB_Bacnet.StartStopCommand_132.bVal := TRUE;
                                    6: 
                                        
                                        FB_Bacnet.StartStopCommand_133.bEnWrite := TRUE;
                                        FB_Bacnet.StartStopCommand_133.bVal := TRUE;
                                    7: 
                                        
                                        FB_Bacnet.StartStopCommand_134.bEnWrite := TRUE;
                                        FB_Bacnet.StartStopCommand_134.bVal := TRUE;
                                    8: 
                                        
                                        FB_Bacnet.StartStopCommand_135.bEnWrite := TRUE;
                                        FB_Bacnet.StartStopCommand_135.bVal := TRUE;
                                    9: 
                                        
                                        FB_Bacnet.StartStopCommand_136.bEnWrite := TRUE;
                                        FB_Bacnet.StartStopCommand_136.bVal := TRUE;
                                    10: 
                                        
                                        FB_Bacnet.StartStopCommand_137.bEnWrite := TRUE;
                                        FB_Bacnet.StartStopCommand_137.bVal := TRUE;
                                    11: 
                                        
                                        FB_Bacnet.StartStopCommand_138.bEnWrite := TRUE;
                                        FB_Bacnet.StartStopCommand_138.bVal := TRUE;
                                    12: 
                                        
                                        FB_Bacnet.StartStopCommand_139.bEnWrite := TRUE;
                                        FB_Bacnet.StartStopCommand_139.bVal := TRUE;
                                    13: 

                                        //FB_Bacnet.StartStopCommand_140.bEnWrite := TRUE;
                                        //FB_Bacnet.StartStopCommand_140.bVal := TRUE;
                                    14: 
                                        
                                        FB_Bacnet.StartStopCommand_141.bEnWrite := TRUE;
                                        FB_Bacnet.StartStopCommand_141.bVal := TRUE;
                                    15: 
                                        
                                        FB_Bacnet.StartStopCommand_142.bEnWrite := TRUE;
                                        FB_Bacnet.StartStopCommand_142.bVal := TRUE;
                                    16: 
                                        
                                        FB_Bacnet.StartStopCommand_143.bEnWrite := TRUE;
                                        FB_Bacnet.StartStopCommand_143.bVal := TRUE;
                                    17: 
                                        
                                        FB_Bacnet.StartStopCommand_144.bEnWrite := TRUE;
                                        FB_Bacnet.StartStopCommand_144.bVal := TRUE;
                                    18: 
                                        
                                        FB_Bacnet.StartStopCommand_145.bEnWrite := TRUE;
                                        FB_Bacnet.StartStopCommand_145.bVal := TRUE;
                                    19: 
                                        
                                        FB_Bacnet.StartStopCommand_146.bEnWrite := TRUE;
                                        FB_Bacnet.StartStopCommand_146.bVal := TRUE;
                                    20: 
                                        
                                        FB_Bacnet.StartStopCommand_147.bEnWrite := TRUE;
                                        FB_Bacnet.StartStopCommand_147.bVal := TRUE;
                                    21: 
                                        
                                        FB_Bacnet.StartStopCommand_148.bEnWrite := TRUE;
                                        FB_Bacnet.StartStopCommand_148.bVal := TRUE;
                                    22: 
                                        
                                        FB_Bacnet.StartStopCommand_176.bEnWrite := TRUE;
                                        FB_Bacnet.StartStopCommand_176.bVal := TRUE;
                                    23: 

                                        //FB_Bacnet.StartStopCommand_177.bEnWrite := TRUE;
                                        //FB_Bacnet.StartStopCommand_177.bVal := TRUE;
                                END_CASE
                            END_IF
                        END_FOR
                    END_IF
                    // Schedule Unit OFF
                    IF wSchedWDHourEndF2_ = currH AND wSchedWDMinEndF2_ = currM AND NOT bUnitTriggered THEN
                        bUnitTriggered := TRUE;
                        FOR i := 1 TO 23 DO
                            // Send command unit OFF
                            IF bUnitF2_[i] THEN 
                                CASE i OF
                                    1: 
                                        
                                        FB_Bacnet.StartStopCommand_128.bEnWrite := TRUE;
                                        FB_Bacnet.StartStopCommand_128.bVal := FALSE;
                                    2: 
                                        
                                        FB_Bacnet.StartStopCommand_129.bEnWrite := TRUE;
                                        FB_Bacnet.StartStopCommand_129.bVal := FALSE;
                                    3: 
                                        
                                        FB_Bacnet.StartStopCommand_130.bEnWrite := TRUE;
                                        FB_Bacnet.StartStopCommand_130.bVal := FALSE;
                                    4: 
                                        
                                        FB_Bacnet.StartStopCommand_131.bEnWrite := TRUE;
                                        FB_Bacnet.StartStopCommand_131.bVal := FALSE;
                                    5: 
                                        
                                        FB_Bacnet.StartStopCommand_132.bEnWrite := TRUE;
                                        FB_Bacnet.StartStopCommand_132.bVal := FALSE;
                                    6: 
                                        
                                        FB_Bacnet.StartStopCommand_133.bEnWrite := TRUE;
                                        FB_Bacnet.StartStopCommand_133.bVal := FALSE;
                                    7: 
                                        
                                        FB_Bacnet.StartStopCommand_134.bEnWrite := TRUE;
                                        FB_Bacnet.StartStopCommand_134.bVal := FALSE;
                                    8: 
                                        
                                        FB_Bacnet.StartStopCommand_135.bEnWrite := TRUE;
                                        FB_Bacnet.StartStopCommand_135.bVal := FALSE;
                                    9: 
                                        
                                        FB_Bacnet.StartStopCommand_136.bEnWrite := TRUE;
                                        FB_Bacnet.StartStopCommand_136.bVal := FALSE;
                                    10: 
                                        
                                        FB_Bacnet.StartStopCommand_137.bEnWrite := TRUE;
                                        FB_Bacnet.StartStopCommand_137.bVal := FALSE;
                                    11: 
                                        
                                        FB_Bacnet.StartStopCommand_138.bEnWrite := TRUE;
                                        FB_Bacnet.StartStopCommand_138.bVal := FALSE;
                                    12: 
                                        
                                        FB_Bacnet.StartStopCommand_139.bEnWrite := TRUE;
                                        FB_Bacnet.StartStopCommand_139.bVal := FALSE;
                                    13: 

                                        //FB_Bacnet.StartStopCommand_140.bEnWrite := TRUE;
                                        //FB_Bacnet.StartStopCommand_140.bVal := FALSE;
                                    14: 
                                        
                                        FB_Bacnet.StartStopCommand_141.bEnWrite := TRUE;
                                        FB_Bacnet.StartStopCommand_141.bVal := FALSE;
                                    15: 
                                        
                                        FB_Bacnet.StartStopCommand_142.bEnWrite := TRUE;
                                        FB_Bacnet.StartStopCommand_142.bVal := FALSE;
                                    16: 
                                        
                                        FB_Bacnet.StartStopCommand_143.bEnWrite := TRUE;
                                        FB_Bacnet.StartStopCommand_143.bVal := FALSE;
                                    17: 
                                        
                                        FB_Bacnet.StartStopCommand_144.bEnWrite := TRUE;
                                        FB_Bacnet.StartStopCommand_144.bVal := FALSE;
                                    18: 
                                        
                                        FB_Bacnet.StartStopCommand_145.bEnWrite := TRUE;
                                        FB_Bacnet.StartStopCommand_145.bVal := FALSE;
                                    19: 
                                        
                                        FB_Bacnet.StartStopCommand_146.bEnWrite := TRUE;
                                        FB_Bacnet.StartStopCommand_146.bVal := FALSE;
                                    20: 
                                        
                                        FB_Bacnet.StartStopCommand_147.bEnWrite := TRUE;
                                        FB_Bacnet.StartStopCommand_147.bVal := FALSE;
                                    21: 
                                        
                                        FB_Bacnet.StartStopCommand_148.bEnWrite := TRUE;
                                        FB_Bacnet.StartStopCommand_148.bVal := FALSE;
                                    22: 
                                        
                                        FB_Bacnet.StartStopCommand_176.bEnWrite := TRUE;
                                        FB_Bacnet.StartStopCommand_176.bVal := FALSE;
                                    23: 

                                        //FB_Bacnet.StartStopCommand_177.bEnWrite := TRUE;
                                        //FB_Bacnet.StartStopCommand_177.bVal := FALSE;
                                END_CASE
                            END_IF
                        END_FOR
                    END_IF
                END_IF
            END_IF

            // Weekend schedule
            IF currD = 0 OR currD = 6 THEN
                IF (wSchedWEHourStartF2_ <> wSchedWEHourEndF2_ OR wSchedWEMinStartF2_ <> wSchedWEMinEndF2_) THEN
                    // Schedule Unit ON
                    IF wSchedWEHourStartF2_ = currH AND wSchedWEMinStartF2_ = currM AND NOT bUnitTriggered THEN
                        bUnitTriggered := TRUE;
                        FOR i := 1 TO 23 DO
                            // Send command unit ON
                            IF bUnitF2_[i] THEN 
                                CASE i OF
                                    1: 
                                        
                                        FB_Bacnet.StartStopCommand_128.bEnWrite := TRUE;
                                        FB_Bacnet.StartStopCommand_128.bVal := TRUE;
                                    2: 
                                        
                                        FB_Bacnet.StartStopCommand_129.bEnWrite := TRUE;
                                        FB_Bacnet.StartStopCommand_129.bVal := TRUE;
                                    3: 
                                        
                                        FB_Bacnet.StartStopCommand_130.bEnWrite := TRUE;
                                        FB_Bacnet.StartStopCommand_130.bVal := TRUE;
                                    4: 
                                        
                                        FB_Bacnet.StartStopCommand_131.bEnWrite := TRUE;
                                        FB_Bacnet.StartStopCommand_131.bVal := TRUE;
                                    5: 
                                        
                                        FB_Bacnet.StartStopCommand_132.bEnWrite := TRUE;
                                        FB_Bacnet.StartStopCommand_132.bVal := TRUE;
                                    6: 
                                        
                                        FB_Bacnet.StartStopCommand_133.bEnWrite := TRUE;
                                        FB_Bacnet.StartStopCommand_133.bVal := TRUE;
                                    7: 
                                        
                                        FB_Bacnet.StartStopCommand_134.bEnWrite := TRUE;
                                        FB_Bacnet.StartStopCommand_134.bVal := TRUE;
                                    8: 
                                        
                                        FB_Bacnet.StartStopCommand_135.bEnWrite := TRUE;
                                        FB_Bacnet.StartStopCommand_135.bVal := TRUE;
                                    9: 
                                        
                                        FB_Bacnet.StartStopCommand_136.bEnWrite := TRUE;
                                        FB_Bacnet.StartStopCommand_136.bVal := TRUE;
                                    10: 
                                        
                                        FB_Bacnet.StartStopCommand_137.bEnWrite := TRUE;
                                        FB_Bacnet.StartStopCommand_137.bVal := TRUE;
                                    11: 
                                        
                                        FB_Bacnet.StartStopCommand_138.bEnWrite := TRUE;
                                        FB_Bacnet.StartStopCommand_138.bVal := TRUE;
                                    12: 
                                        
                                        FB_Bacnet.StartStopCommand_139.bEnWrite := TRUE;
                                        FB_Bacnet.StartStopCommand_139.bVal := TRUE;
                                    13: 
                                        //FB_Bacnet.StartStopCommand_140.bEnWrite := TRUE;
                                        //FB_Bacnet.StartStopCommand_140.bVal := TRUE;
                                    14: 
                                        
                                        FB_Bacnet.StartStopCommand_141.bEnWrite := TRUE;
                                        FB_Bacnet.StartStopCommand_141.bVal := TRUE;
                                    15: 
                                        
                                        FB_Bacnet.StartStopCommand_142.bEnWrite := TRUE;
                                        FB_Bacnet.StartStopCommand_142.bVal := TRUE;
                                    16: 
                                        
                                        FB_Bacnet.StartStopCommand_143.bEnWrite := TRUE;
                                        FB_Bacnet.StartStopCommand_143.bVal := TRUE;
                                    17: 
                                        
                                        FB_Bacnet.StartStopCommand_144.bEnWrite := TRUE;
                                        FB_Bacnet.StartStopCommand_144.bVal := TRUE;
                                    18: 
                                        
